// TIA Portal project "OVEN" (V18)

(* hardware
DEVICE "S7-1200-Station_1"  S7-1200 Station
   slot 0: "Baugruppenträger_0"  S7-1200 Rack  Rack  V1.0
   slot 1: "OVEN"  CPU 1215C DC/DC/DC  6ES7 215-1AG40-0XB0  V4.5
*)

// ===== PLC "OVEN"  CPU 1215C DC/DC/DC =====

VAR_GLOBAL   // PLC tag table "Standard-Variablentabelle"
   "sauger_vorn" AT %I0.0 : Bool;
   "sauger_hinten" AT %I0.1 : Bool;
   "lichtschranke" AT %I0.2 : Bool;
   "ofenschieber_innen" AT %I0.3 : Bool;
   "ofenschieber_außen" AT %I0.4 : Bool;
   "sauger_rein" AT %Q0.0 : Bool;
   "sauger_raus" AT %Q0.1 : Bool;
   "ofenschieber_rein" AT %Q0.2 : Bool;
   "ofenschieber_raus" AT %Q0.3 : Bool;
   "kompressor" AT %Q0.4 : Bool;
   "lampe_ofen" AT %Q0.5 : Bool;
   "vakuum" AT %Q0.6 : Bool;
   "sauger_senken" AT %Q0.7 : Bool;
   "ofentür" AT %Q1.0 : Bool;
   "pwm_sauger" AT %Q1.1 : Bool;
END_VAR

DATA_BLOCK "LOOP_DB"   // DB2
{ S7_Optimized_Access := 'TRUE' }
VERSION : 0.1
// stored: InstanceOfName LOOP
"LOOP"
BEGIN
END_DATA_BLOCK

FUNCTION_BLOCK "LOOP"   // FB1, SCL
{ S7_Optimized_Access := 'TRUE' }
VERSION : 0.1
   VAR
      model : String := 'OVEN';
      idle : Bool;
      pick : Bool;
      drop : Bool;
      fire : Bool;
      duration : Int := 5;
      pick_finished : Bool;
      drop_finished : Bool;
      fire_finished : Bool;
      pick_failed : Bool;
      drop_failed : Bool;
      drop_aktiv : Bool;
      pick_aktiv : Bool;
      fire_aktiv : Bool;
      "step" : Int;
      warte_start : Bool;
      warte_zeit : Time;
      warte : TON_TIME;
   END_VAR
   VAR RETAIN
      zeit_prozessende : Time := T#2S;
      zeit_saugerRunter : Time := T#850MS;
      zeit_vakuum_loesen : Time := T#1S;
   END_VAR
   VAR
      "version" : String := '1.3.0';
   END_VAR
BEGIN
   #warte.TON(IN:=#warte_start,
                        PT:=#warte_zeit);

   CASE #step OF
       0:  // Init
           #idle := TRUE;
           #drop_failed := FALSE;
           #pick_failed := FALSE;
           #drop_failed := FALSE;
           #fire_finished := FALSE;
           #pick_finished := FALSE;
           #drop_finished := FALSE;
           #step := 1;
       1: // erwartet befehle
           IF #pick THEN
               #pick_aktiv := TRUE;
               #idle := FALSE;
               #pick := FALSE;
               #step := 10;
           ELSIF #drop THEN
               #drop_aktiv := TRUE;
               #idle := FALSE;
               #drop := FALSE;
               #step := 50;
           ELSIF #fire THEN
               #fire_aktiv := TRUE;
               #idle := FALSE;
               #fire := FALSE;
               #step := 100;
           END_IF
           ;
       200: // ENDE jedes Prozesses
           "vakuum" := FALSE;
           "kompressor" := FALSE;
           "pwm_sauger" := FALSE;
           "sauger_raus" := FALSE;
           "sauger_rein" := FALSE;
           #warte_zeit := #zeit_prozessende;
           #warte_start := TRUE;
           IF #warte.Q THEN
               #warte_start := FALSE;
               #step := 0;
           END_IF
           ;
       10: // ---------------------------- Start PICK
           // check ob ofenschieber draußen
           IF "ofenschieber_außen" THEN
               #step := 14;
           END_IF;
           // kompressor an kurz warten
           "kompressor" := TRUE;
           #warte_zeit := T#200ms;
           #warte_start := TRUE;
           IF #warte.Q THEN
               #warte_start := FALSE;
               #step := 11;
           END_IF
           ;
       11: // ofentür auf kurz warten
           "ofentür" := TRUE;
           #warte_zeit := T#200ms;
           #warte_start := TRUE;
           IF #warte.Q THEN
               #warte_start := FALSE;
               #step := 12;
           END_IF
           ;
       12: // ofenschieber raus
           "ofenschieber_raus" := TRUE;
           IF "ofenschieber_außen" THEN
               "ofenschieber_raus" := FALSE;
               #step := 13;
           END_IF
           ;
       13 : // ofentür zu
           "ofentür" := FALSE;
           "kompressor" := FALSE;
           #step := 14
           ;
       14: // sauger raus
           "pwm_sauger" := TRUE;
           "sauger_raus" := TRUE;
           IF "sauger_vorn" THEN
               "sauger_raus" := FALSE;
               #step := 15;
           END_IF
           ;
       15: // kompressor an kurz warten
           "kompressor" := TRUE;
           #warte_zeit := T#200ms;
           #warte_start := TRUE;
           IF #warte.Q THEN
               #warte_start := FALSE;
               #step := 16;
           END_IF
           ;
       16: // sauger runter
           "sauger_senken" := TRUE;
           #warte_zeit := #zeit_saugerRunter;
           #warte_start := TRUE;
           IF #warte.Q THEN
               #warte_start := FALSE;
               "vakuum" := TRUE;
               #step := 17;
           END_IF
           ;
       17: // kurz warten sauger hoch
           #warte_zeit := T#300ms;
           #warte_start := TRUE;
           IF #warte.Q THEN
               "sauger_senken" := FALSE;
               #warte_start := FALSE;
               #step := 18;
           END_IF
           ;
       18: // sauger rein
           "sauger_rein" := TRUE;
           IF "sauger_hinten" THEN
               "sauger_rein" := FALSE;
               #step := 19;
           END_IF
           ;
       19: // kurz warten
           #warte_zeit := T#300ms;
           #warte_start := TRUE;
           IF #warte.Q THEN
               #warte_start := FALSE;
               #step := 20;
           END_IF
           ;
       20: // check pick
           IF "lichtschranke" THEN
               #pick_failed := TRUE;
               #step := 30; // zu Prozess Ende
           ELSE
               #step := 21
                 ;
           END_IF
           ;
       21: // sauger runter 
           "sauger_senken" := TRUE;
           #warte_zeit := #zeit_saugerRunter;
           #warte_start := TRUE;
           IF #warte.Q THEN
               #warte_start := FALSE;
               #step := 22;
           END_IF
           ;
       22: // Vakuum lösen kurz
           "vakuum" := FALSE;
           #warte_zeit := #zeit_vakuum_loesen;
           #warte_start := TRUE;
           IF #warte.Q THEN
               "sauger_senken" := FALSE;
               #warte_start := FALSE;
               #step := 30;
           END_IF
           ;
       30: // Prozessende
           IF #pick_failed THEN
               #pick_aktiv := FALSE;
           ELSE
               #pick_aktiv := FALSE;
               #pick_finished := TRUE;
           END_IF;
           #step := 200
           ;
           // ---------------------------- END PICK ----------------------------




       50: // ---------------------------- Start DROP
           // kompressor an kurz warten
           "pwm_sauger" := TRUE;
           "kompressor" := TRUE;
           #warte_zeit := T#200ms;
           #warte_start := TRUE;
           IF #warte.Q THEN
               #warte_start := FALSE;
               #step := 51;
           END_IF
           ;
       51: // sauger runter kurz warten
           "sauger_senken" := TRUE;
           #warte_zeit := #zeit_saugerRunter;
           #warte_start := TRUE;
           IF #warte.Q THEN
               #warte_start := FALSE;
               "vakuum" := TRUE;
               #step := 52;
           END_IF
           ;
       52: // kurz warten sauger hoch
           #warte_zeit := T#100ms;
           #warte_start := TRUE;
           IF #warte.Q THEN
               "sauger_senken" := FALSE;
               #warte_start := FALSE;
               #step := 70;
           END_IF
           ;
       70: // warte Zeit
           #warte_zeit := T#500ms;
           #warte_start := TRUE;
           IF #warte.Q THEN
               #warte_start := FALSE;
               #step := 71;
           END_IF
           ;
       71: // Drop Check
           IF "lichtschranke" THEN
               #drop_failed := TRUE;
               #step := 58; // zu prozess Ende
           ELSE
               #step := 53; // normal weiter
           END_IF
           ;

       53: // sauger raus
           "sauger_raus" := TRUE;
           IF "sauger_vorn" THEN
               "sauger_raus" := FALSE;
               #step := 54;
           END_IF
           ;
       54: // sauger runter kurz warten
           "sauger_senken" := TRUE;
           #warte_zeit := #zeit_saugerRunter;
           #warte_start := TRUE;
           IF #warte.Q THEN
               #warte_start := FALSE;
               #step := 55;
           END_IF
           ;
       55: // Vakuum lösen kurz warten und sauger hoch
           "vakuum" := FALSE;
           #warte_zeit := #zeit_vakuum_loesen;
           #warte_start := TRUE;
           IF #warte.Q THEN
               "sauger_senken" := FALSE;
               #warte_start := FALSE;
               #step := 56;
           END_IF
           ;
       56: // kompressor aus, kurz warten
           "kompressor" := FALSE;
           #warte_zeit := T#200ms;
           #warte_start := TRUE;
           IF #warte.Q THEN
               #warte_start := FALSE;
               #step := 57;
           END_IF
           ;
       57: // sauger rein
           "sauger_rein" := TRUE;
           IF "sauger_hinten" THEN
               "sauger_rein" := FALSE;
               #step := 58;
           END_IF
           ;
       58: // Prozess Ende
           IF #drop_failed THEN
               #drop_aktiv := FALSE;
           ELSE
               #drop_aktiv := FALSE;
               #drop_finished := TRUE;
           END_IF;
           #step := 200;
           ;
       100: // ---------------------------- Start FIRE ----------------------------
           // kompressor an kurz warten
           "kompressor" := TRUE;
           #warte_zeit := T#200ms;
           #warte_start := TRUE;
           IF #warte.Q THEN
               #warte_start := FALSE;
               #step := 101;
           END_IF
           ;
       101: // ofentür auf
           "ofentür" := TRUE;
           #warte_zeit := T#200ms;
           #warte_start := TRUE;
           IF #warte.Q THEN
               #warte_start := FALSE;
               #step := 102;
           END_IF
           ;
       102: // ofenschieber rein
           "ofenschieber_rein" := TRUE;
           IF "ofenschieber_innen" THEN
               "ofenschieber_rein" := FALSE;
               #step := 103;
           END_IF
           ;
       103 : // ofentür zu
           "ofentür" := FALSE;
           "kompressor" := FALSE;
           #step := 104
           ;
       104: // BRENNE
           "lampe_ofen" := TRUE;
           #warte_zeit := T#1s * #duration;
           #warte_start := TRUE;
           IF #warte.Q THEN
               #warte_start := FALSE;
               "lampe_ofen" := FALSE;
               #step := 105;
           END_IF
           ;
       105: // kurz warten (abkühlen)
           #warte_zeit := T#1000ms;
           #warte_start := TRUE;
           IF #warte.Q THEN
               #warte_start := FALSE;
               #step := 106;
           END_IF
           ;
       106: // kompressor an kurz warten
           "kompressor" := TRUE;
           #warte_zeit := T#200ms;
           #warte_start := TRUE;
           IF #warte.Q THEN
               #warte_start := FALSE;
               #step := 108;
           END_IF
           ;
       108: // ofentür auf kurz warten
           "ofentür" := TRUE;
           #warte_zeit := T#200ms;
           #warte_start := TRUE;
           IF #warte.Q THEN
               #warte_start := FALSE;
               #step := 109;
           END_IF
           ;
       109: // ofenschieber raus
           "ofenschieber_raus" := TRUE;
           IF "ofenschieber_außen" THEN
               "ofenschieber_raus" := FALSE;
               #step := 110;
           END_IF
           ;
       110: // ofentür zu
           "ofentür" := FALSE;
           "kompressor" := FALSE;
           #step := 111
           ;
       111:// kurz warten
           #fire_aktiv := FALSE;
           #fire_finished := TRUE;
           #step := 200;
           // ---------------------------- END FIRE 
       ELSE  // Statement section ELSE
           ;
   END_CASE;
END_FUNCTION_BLOCK

ORGANIZATION_BLOCK "Main"   // OB1, LAD, ProgramCycle
TITLE = "Main Program Sweep (Cycle)"
{ S7_Optimized_Access := 'TRUE' }
VERSION : 0.1
   VAR_INPUT
      Initial_Call : Bool;   // Initial call of this OB
      Remanence : Bool;   // =True, if remanent data are available
   END_VAR
BEGIN

REGION Network 1
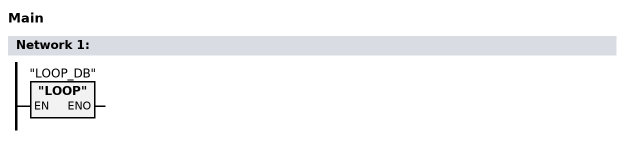
   RUNG wire#powerrail
      "LOOP_DB"()
   END_RUNG
   // the same network as SCL:
   "LOOP_DB"();   // "LOOP"
END_REGION
END_ORGANIZATION_BLOCK